// TIA Portal V17 export
// export: Created 2023-04-07T15:33:28.3575336Z, ExportSetting WithDefaults, DisplayName Totally Integrated Automation Portal, DisplayVersion V17 Update 4, DisplayName TIA Portal Openness, DisplayVersion V17 Update 4, DisplayName TIA Portal Version Control Interface, DisplayVersion V17, DisplayName STEP 7 Professional, DisplayVersion V17 Update 4, DisplayName STEP 7 Safety, DisplayVersion V17, DisplayName WinCC Professional, DisplayVersion V17 Update 4
DATA_BLOCK "SM1"   // DB61
{ S7_Optimized_Access := 'TRUE' }
VERSION : 0.1
// stored: AutoNumber false, DBAccessibleFromOPCUA true, DBAccessibleFromWebserver true, IsOnlyStoredInLoadMemory false, IsRetainMemResEnabled false, IsWriteProtectedInAS false, MemoryReserve 100
   VAR
      xT11 : Bool;
      xT21 : Bool;
      xT22 : Bool;
      xT31 : Bool;
      xT32 : Bool;
      xT33 : Bool;
      xT34 : Bool;
      xT41 : Bool;
      xT42 : Bool;
      xT43 : Bool;
      xT44 : Bool;
      xT51 : Bool;
      xT52 : Bool;
      xT53 : Bool;
      xT61 : Bool;
      xT62 : Bool;
      xT71 : Bool;
      xT72 : Bool;
      xT73 : Bool;
      xT74 : Bool;
      xT75 : Bool;
      xT76 : Bool;
      xT81 : Bool;
      xT91 : Bool;
      xSsBootSt : Bool;
      xSsWarmUpSt : Bool;
      xSsReadySt : Bool;
      xSsStandBySt : Bool;
      xSsRunSt : Bool;
      xSsTestSt : Bool;
      xSsAutoMaintSt : Bool;
      xSsStopSt : Bool;
      xSsFaultSt : Bool;
      iCountSS : Int;
      xBootSt : Bool;
      xRunPlcSt : Bool;
      xCommCmd : Bool;
      xAuxCmd : Bool;
      xCommSt : Bool;
      xAuxSt : Bool;
      xFltSt : Bool;
      xEnbSSysSt : Bool;
      xReadyCondSt : Bool;
      xTestCmd : Bool;
      xBattCloseCmd : Bool;
      xBattCloseSt : Bool;
      xBattOpenSt : Bool;
      xStopCmd : Bool;
      xStandByCmd : Bool;
      xAutomaintCmd : Bool;
      xStopAutomaintCmd : Bool;
      xAutomaintSt : Bool;
      xRunCmd : Bool;
      xPCSenbCmd : Bool;
      xPCSrunCmd : Bool;
      xMVbreakerCloseSt : Bool;
      xPCSrunSt : Bool;
      xPCSstopSt : Bool;
      xPCSreadySt : Bool;
      rPacAutomRef : Real;
      xVacPCS : Bool;
      xMVbreakerOpenCmd : Bool;
      xMVbreakerOpenSt : Bool;
   END_VAR
BEGIN
END_DATA_BLOCK
